// TIA Portal V20 export
VAR_GLOBAL   // PLC tag table "1.Entrada Digital"
   Input_1 AT %I0.0 : Bool;
   Input_2 AT %I0.1 : Bool;
   Input_3 AT %I0.2 : Bool;
   Input_4 AT %I0.3 : Bool;
   Input_5 AT %I0.4 : Bool;
   Input_6 AT %I0.5 : Bool;
   Input_7 AT %I0.6 : Bool;
   Input_8 AT %I0.7 : Bool;
   Input_9 AT %I1.0 : Bool;
   Input_10 AT %I1.1 : Bool;
   Input_11 AT %I1.2 : Bool;
   Input_12 AT %I1.3 : Bool;
   Input_13 AT %I1.4 : Bool;
   Input_14 AT %I1.5 : Bool;
   Input_15 AT %I1.6 : Bool;
   Input_16 AT %I1.7 : Bool;
END_VAR
